TEXTLIST stAlarmEventData_TextList
  0 = ''
  1 = 'Maintenance'
  2 = 'Message'
  3 = 'Hint'
  4 = 'StateInfo'
  5 = 'Instruction'
  6 = 'Warning'
  7 = 'Alarm'
  8 = 'Parameter'
   = ''
END_TEXTLIST

(* stored: Version 1.1.0.1
   TextList stAlarmEventData_TextList: Id {55d16c12-cc99-4460-ac4c-323441edcdd0} *)
